{attribute 'qualified_only'}
{attribute 'strict'}
TYPE DUT_ENUM_TEST :
(
	zeroeth_member := 0,
	first_member := 1,
	second_member := 2,
	third_member := 3
);
END_TYPE

(* stored: Version 1.1.0.1, ProductVersion 3.1.4022.10
   DUT DUT_ENUM_TEST: Id {cf358361-ca0c-4f8d-a342-4d03831ebeec} *)
